ABB RobotStudio station: practica3.rspag

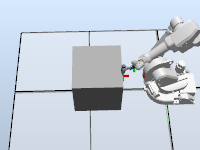
--- station ---
Station practica3 (saved by RobotStudio 20.4.9280.0)
Controller Controlador4
  mechanical unit ROB_1: IRB1600_6_145__02, 6 joints, base frame (0, 0, 0) mm
Layout (positions relative to the parent item):
  - IRB1600_6_145__02 [mechanism, from Robots\IRB1600_6_145_G_02.rslib] at (0, 0, 0) mm; joint values [0.326, -0.2862, 0.8219, -0.4788, 0.4423, 0.699] (rad or m)
  - MyTool [mechanism, from Training Objects\myTool.rslib] at (483.67, 150, 800.53) mm, rotated rx -180 ry 38 rz -180 deg
  - Pieza_1 [part]
Attachment: MyTool is attached to IRB1600_6_145__02 / Link6
Targets, tools, work objects and paths stored in the station and not in the controller backup, written as RAPID:
! task T_ROB1
MODULE Module1
  PROC Path_10()
    MoveL pInicio,v1000,z100,MyTool\WObj:=wobj0;
  ENDPROC
ENDMODULE


--- Backups/Controlador4/RAPID/TASK1/PROGMOD/CalibData.mod ---
MODULE CalibData
    PERS tooldata MyTool:=[TRUE,[[31.792631019,0,229.638935148],[0.945518576,0,0.325568154,0]],[1,[0,0,1],[1,0,0,0],0,0,0]];
ENDMODULE

--- Backups/Controlador4/RAPID/TASK1/PROGMOD/Module1.mod ---
MODULE Module1
        CONST robtarget pInicio:=[[600,150,600],[0,0,1,0],[0,0,0,0],[9E+09,9E+09,9E+09,9E+09,9E+09,9E+09]];
!***********************************************************
    !
    ! Módulo:  Module1
    !
    ! Descripción:
    !   <Introduzca la descripción aquí>
    !
    ! Autor: franc
    !
    ! Versión: 1.0
    !
    !***********************************************************


    !***********************************************************
    !
    ! Procedimiento Main
    !
    !   Este es el punto de entrada de su programa
    !
    !***********************************************************
    PROC main()
        !Añada aquí su código
        MoveL pInicio,v100,z0,MyTool\WObj:=wobj0;
        Senoide pInicio, 150, 100;
        MoveL pInicio,v100,z0,MyTool\WObj:=wobj0;

    ENDPROC

    PROC Senoide(robtarget pIni, num amplX, num amplY)

        CONST num nPuntos := 100+1;
        VAR robtarget tabPos{nPuntos}; !Array de puntos
        VAR num posX;
        VAR num posY;
        VAR num incr;
        VAR robtarget pApoyo;
        !Variables para la rotacion de la pieza
        VAR num angX;
        VAR num angY;
        VAR num angZ;
        VAR robtarget pAux;
        VAR num hipotenusa;
        VAR num CatOp;
        VAR num CatCo;
        VAR num posY2;
        VAR num seno;
        VAR num angulo;

        !Añadimos el punto inicial
        tabPos{1} := pIni; ! Punto inicial añadido a la tabla de puntos

        !Calculamos el incremento
        incr := (amplX*2) / nPuntos;

        !Inicializamos
        posY2 := 0;

        !Creamos la tabla de puntos
        FOR i FROM 2 TO nPuntos DO ! Empieza en 0 o 1 ( empezamos en 1 porque el 0 será la posición inicial)
            !funcion seno
            posX := ((i*incr) * 360) / (amplX * 2); !Angulo que le pasamos al seno
            posY := amplY * Sin(posX); !Calculamos la altura de Y según su posicion en el eje X (calculado el angulo previamente posX)

            pApoyo := Offs (pIni, incr * (i - 2), posY, 0); !Hacemos el punto

            !Calculamos la hipotenusa, el cateto contiguo y el cateto opuesto
            CatCo := incr;
            CatOp := posY - posY2; !Y actual - anterior
            posY2 := posY; !Actualizamos el valor anterior al actual
            hipotenusa := Sqrt((CatCo * CatCo) + (CatOp * CatOp));

            !Sacamos el seno para sacarle el angulo haciendo arcoseno
            seno := CatOp / hipotenusa;
            angulo := ASin(seno);

            !Sacamos el cuaternio de EulerZXY()
            angZ := EulerZYX(\Z, pApoyo.rot);
            angY := EulerZYX(\Y, pApoyo.rot);
            angX := EulerZYX(\X, pApoyo.rot);

            !Guardamos la rotación de los puntos
            pAux := pApoyo;
            pAux.rot := OrientZYX(angZ + angulo,angY,angX);

            tabPos{i} := pAux; !Guadamos el punto en la tabla


        ENDFOR

        !Recorremos la tabla de puntos
        FOR i FROM 1 TO nPuntos DO

            !Movemos el brazo
            MoveL tabPos{i},v100,z0,MyTool\WObj:=wobj0;
        ENDFOR

    ENDPROC
ENDMODULE
